# EPICS autosave request: support/ip/2-9/ipApp/Db/Keithley2kDMM_channelN_settings.req
#FILE... Keithley2kDMM_channelN_settings.req
#USAGE... Keithley2kDMM.db fields autosave'd.
$(P)$(Dmm)$(Ch)_on_off.VAL
$(P)$(Dmm)$(Ch)_raw.DESC
$(P)$(Dmm)$(Ch)_calc.DESC
$(P)$(Dmm)$(Ch)_calc.PREC
$(P)$(Dmm)$(Ch)_calc.SCAN
$(P)$(Dmm)$(Ch)_calc.INAN
$(P)$(Dmm)$(Ch)_calc.INBN
$(P)$(Dmm)$(Ch)_calc.INCN
$(P)$(Dmm)$(Ch)_calc.INDN
$(P)$(Dmm)$(Ch)_calc.INEN
$(P)$(Dmm)$(Ch)_calc.INFN
$(P)$(Dmm)$(Ch)_calc.INGN
$(P)$(Dmm)$(Ch)_calc.INHN
$(P)$(Dmm)$(Ch)_calc.ININ
$(P)$(Dmm)$(Ch)_calc.INJN
$(P)$(Dmm)$(Ch)_calc.INKN
$(P)$(Dmm)$(Ch)_calc.INLN
$(P)$(Dmm)$(Ch)_calc.B
$(P)$(Dmm)$(Ch)_calc.C
$(P)$(Dmm)$(Ch)_calc.D
$(P)$(Dmm)$(Ch)_calc.E
$(P)$(Dmm)$(Ch)_calc.F
$(P)$(Dmm)$(Ch)_calc.G
$(P)$(Dmm)$(Ch)_calc.H
$(P)$(Dmm)$(Ch)_calc.I
$(P)$(Dmm)$(Ch)_calc.J
$(P)$(Dmm)$(Ch)_calc.K
$(P)$(Dmm)$(Ch)_calc.L
$(P)$(Dmm)$(Ch)_calc.CALC
$(P)$(Dmm)$(Ch)_calc.INAP
$(P)$(Dmm)$(Ch)_calc.INBP
$(P)$(Dmm)$(Ch)_calc.INCP
$(P)$(Dmm)$(Ch)_calc.INDP
$(P)$(Dmm)$(Ch)_calc.INEP
$(P)$(Dmm)$(Ch)_calc.INFP
$(P)$(Dmm)$(Ch)_calc.INGP
$(P)$(Dmm)$(Ch)_calc.INHP
$(P)$(Dmm)$(Ch)_calc.INIP
$(P)$(Dmm)$(Ch)_calc.INJP
$(P)$(Dmm)$(Ch)_calc.INKP
$(P)$(Dmm)$(Ch)_calc.INLP
$(P)$(Dmm)$(Ch)_calc.DOLN
$(P)$(Dmm)$(Ch)_calc.OUTN
$(P)$(Dmm)$(Ch)_calc.SCAN
